// TIA Portal V19 export
DATA_BLOCK "Area02_Messages"   // DB173
// stored: MemoryReserve 100
   VAR
      "A" : Struct
         Msg : Array[1..576] of Bool;
         Hmi : Array[1..36] of Word;
         Ack : Array[1..36] of Word;
      END_STRUCT;
      W : Struct
         Msg : Array[1..384] of Bool;
         Hmi : Array[1..24] of Word;
         Ack : Array[1..24] of Word;
      END_STRUCT;
   END_VAR
BEGIN
   // "A".Msg[2] : h
   // "A".Msg[3] : hsfdd
END_DATA_BLOCK
